FUNCTION_BLOCK CHECKPOINT_DATA_PUBLISHER (* Composite Function Block Type *)
  (* Standard: 61499-2 *)
  (* Version 0.0, 12/17/2022, Dmitrii, Flexbridge AB, template *)
  PACKAGE UAO.Hackathon;
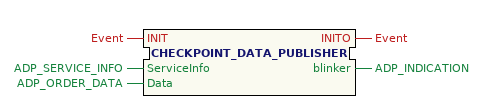
  EVENT_INPUT
    INIT;
  END_EVENT
  EVENT_OUTPUT
    INITO;
  END_EVENT
  SOCKETS
    ServiceInfo : ADP_SERVICE_INFO;
    Data : ADP_ORDER_DATA;
  END_SOCKETS
  PLUGS
    blinker : ADP_INDICATION;
  END_PLUGS
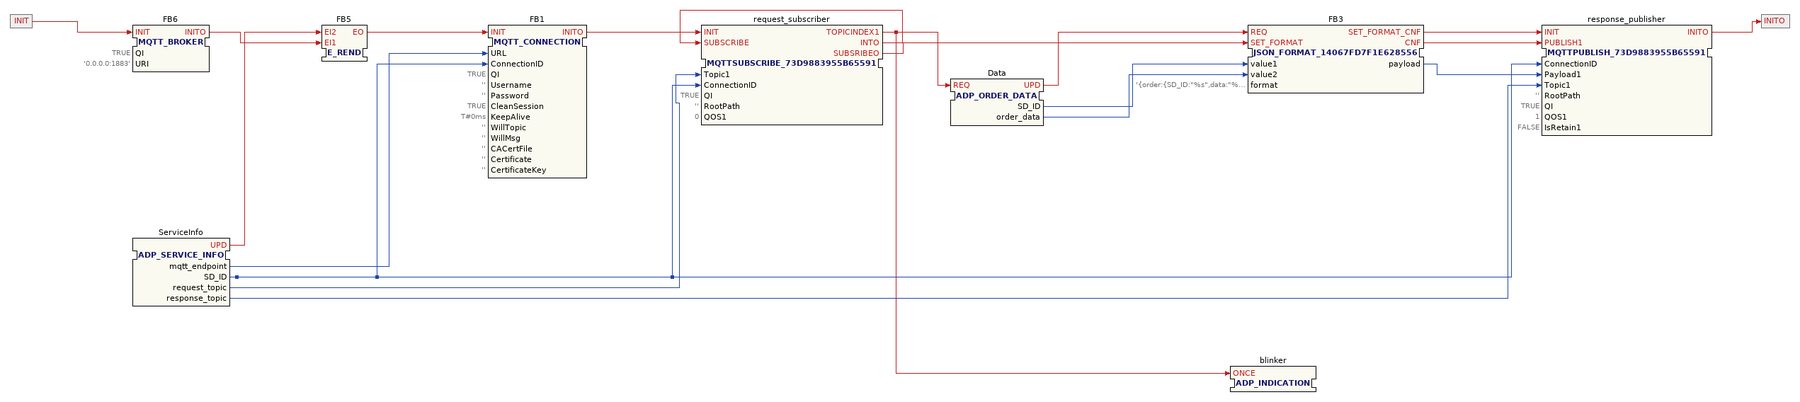
  (* Here subscriber could be checking for a specific request from 'RecPayload1', i.e. "GET" *)
  FBS
    FB1 : MQTT_CONNECTION(QI := TRUE, Username := '', Password := '', CleanSession := TRUE, KeepAlive := T#0ms, WillTopic := '', WillMsg := '', CACertFile := '', Certificate := '', CertificateKey := '');
    response_publisher : MQTTPUBLISH_73D9883955B65591(RootPath := '', QI := TRUE, QOS1 := 1, IsRetain1 := FALSE); {SET_ATTRIBUTE(Configuration.GenericFBType.InterfaceParams, nxtControl.CommProtocols#CNTX:=1)}
    FB3 : JSON_FORMAT_14067FD7F1E628556(format := '{order:{SD_ID:"%s",data:"%s"}}'); {SET_ATTRIBUTE(Configuration.GenericFBType.InterfaceParams, Runtime.Base#CNT:=2;value${CNT$}:STRING,STRING)}
    request_subscriber : MQTTSUBSCRIBE_73D9883955B65591(QI := TRUE, RootPath := '', QOS1 := 0); {SET_ATTRIBUTE(Configuration.GenericFBType.InterfaceParams, nxtControl.CommProtocols#CNTX:=1)}
    FB5 : E_REND;
    FB6 : MQTT_BROKER(QI := TRUE, URI := '0.0.0.0:1883');
  END_FBS
  EVENT_CONNECTIONS
    Data.UPD TO FB3.REQ;
    FB1.INITO TO request_subscriber.INIT;
    FB3.SET_FORMAT_CNF TO response_publisher.INIT;
    FB3.CNF TO response_publisher.PUBLISH1;
    ServiceInfo.UPD TO FB5.EI2;
    FB5.EO TO FB1.INIT;
    response_publisher.INITO TO INITO;
    INIT TO FB6.INIT;
    FB6.INITO TO FB5.EI1;
    request_subscriber.TOPICINDEX1 TO Data.REQ;
    request_subscriber.INTO TO request_subscriber.SUBSCRIBE;
    request_subscriber.SUBSRIBEO TO FB3.SET_FORMAT;
    request_subscriber.TOPICINDEX1 TO blinker.ONCE;
  END_CONNECTIONS
  DATA_CONNECTIONS
    ServiceInfo.mqtt_endpoint TO FB1.URL;
    ServiceInfo.SD_ID TO FB1.ConnectionID;
    ServiceInfo.SD_ID TO response_publisher.ConnectionID;
    FB3.payload TO response_publisher.Payload1;
    Data.SD_ID TO FB3.value1;
    Data.order_data TO FB3.value2;
    ServiceInfo.request_topic TO request_subscriber.Topic1;
    ServiceInfo.response_topic TO response_publisher.Topic1;
    ServiceInfo.SD_ID TO request_subscriber.ConnectionID;
  END_CONNECTIONS
END_FUNCTION_BLOCK
